// Mitsubishi GX Works2 project: timer4   PLC: Q03UDV

PROGRAM MAIN
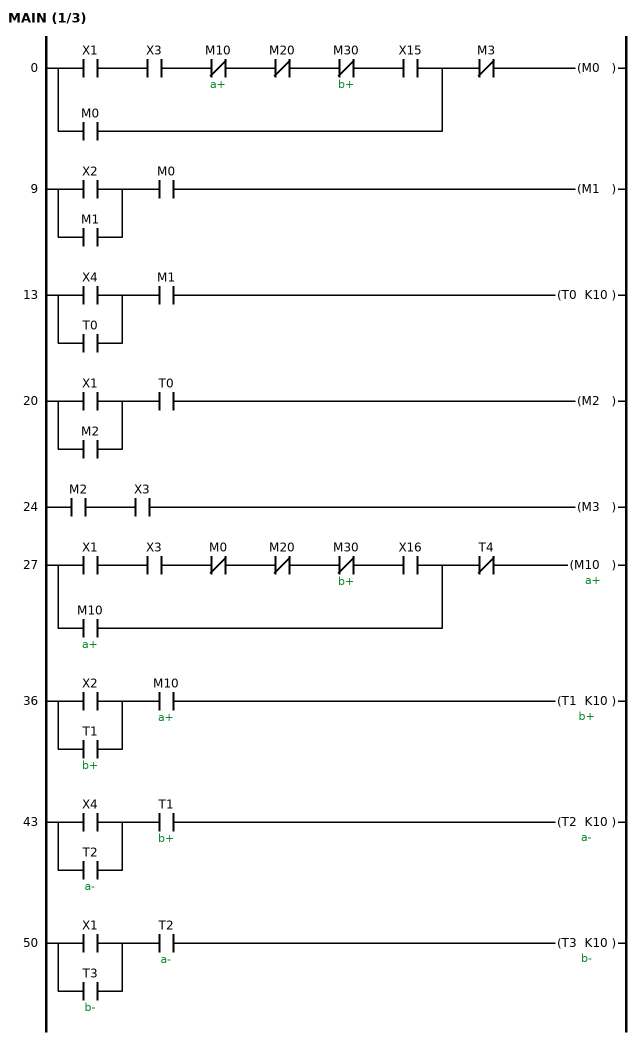
0     LD      X1
      AND     X3
      ANI     M10  ; a+
      ANI     M20
      ANI     M30  ; b+
      AND     X15
      OR      M0
      ANI     M3
      OUT     M0
9     LD      X2
      OR      M1
      AND     M0
      OUT     M1
13    LD      X4
      OR      T0
      AND     M1
      OUT     T0 K10
20    LD      X1
      OR      M2
      AND     T0
      OUT     M2
24    LD      M2
      AND     X3
      OUT     M3
27    LD      X1
      AND     X3
      ANI     M0
      ANI     M20
      ANI     M30  ; b+
      AND     X16
      OR      M10  ; a+
      ANI     T4
      OUT     M10  ; a+
36    LD      X2
      OR      T1  ; b+
      AND     M10  ; a+
      OUT     T1 K10  ; b+
43    LD      X4
      OR      T2  ; a-
      AND     T1  ; b+
      OUT     T2 K10  ; a-
50    LD      X1
      OR      T3  ; b-
      AND     T2  ; a-
      OUT     T3 K10  ; b-
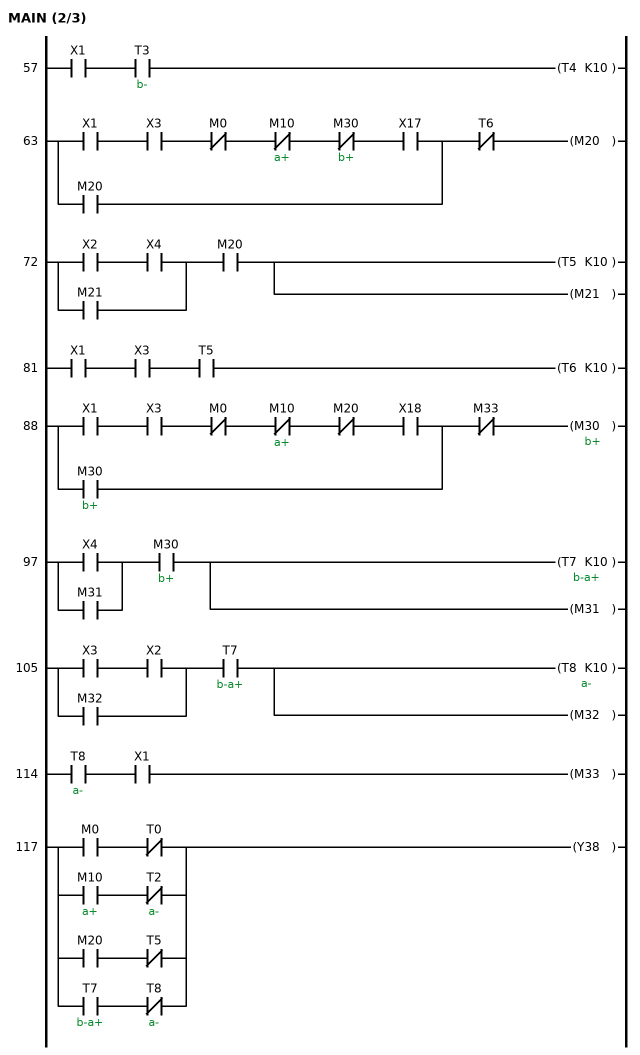
57    LD      X1
      AND     T3  ; b-
      OUT     T4 K10
63    LD      X1
      AND     X3
      ANI     M0
      ANI     M10  ; a+
      ANI     M30  ; b+
      AND     X17
      OR      M20
      ANI     T6
      OUT     M20
72    LD      X2
      AND     X4
      OR      M21
      AND     M20
      OUT     T5 K10
      OUT     M21
81    LD      X1
      AND     X3
      AND     T5
      OUT     T6 K10
88    LD      X1
      AND     X3
      ANI     M0
      ANI     M10  ; a+
      ANI     M20
      AND     X18
      OR      M30  ; b+
      ANI     M33
      OUT     M30  ; b+
97    LD      X4
      OR      M31
      AND     M30  ; b+
      OUT     T7 K10  ; b-a+
      OUT     M31
105   LD      X3
      AND     X2
      OR      M32
      AND     T7  ; b-a+
      OUT     T8 K10  ; a-
      OUT     M32
114   LD      T8  ; a-
      AND     X1
      OUT     M33
117   LD      M0
      ANI     T0
      LD      M10  ; a+
      ANI     T2  ; a-
      ORB
      LD      M20
      ANI     T5
      ORB
      LD      T7  ; b-a+
      ANI     T8  ; a-
      ORB
      OUT     Y38
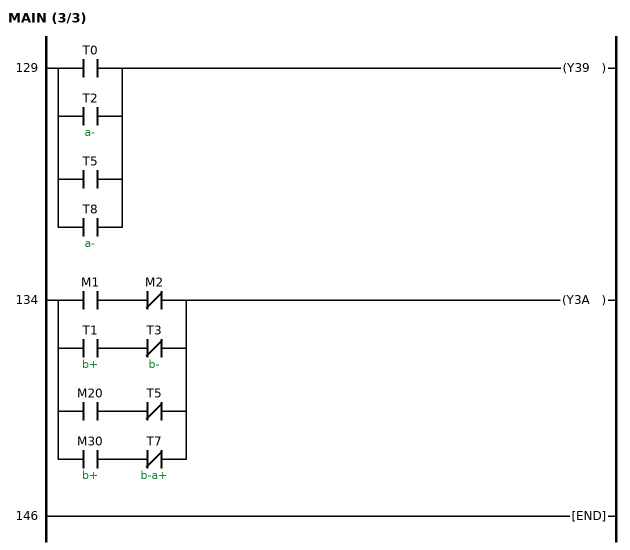
129   LD      T0
      OR      T2  ; a-
      OR      T5
      OR      T8  ; a-
      OUT     Y39
134   LD      M1
      ANI     M2
      LD      T1  ; b+
      ANI     T3  ; b-
      ORB
      LD      M20
      ANI     T5
      ORB
      LD      M30  ; b+
      ANI     T7  ; b-a+
      ORB
      OUT     Y3A
146   END
END_PROGRAM
